{attribute wpf [Container(Layout.Stack)]}
FUNCTION_BLOCK TcoEmergencyStop EXTENDS TcoElements.TcoDi
VAR_OUTPUT
END_VAR
VAR
END_VAR

SUPER^(inoSignal:=inoSignal);
IF inoSignal THEN
	Messenger.Error('<#Emergency stop active#>').Pin();
END_IF;

END_FUNCTION_BLOCK

(* stored: Version 1.1.0.1
   POU TcoEmergencyStop: Id {83bdb684-36b8-4905-8497-ac18239f9927}, SpecialFunc None *)
